# EPICS autosave request: pixciApp/Db/Pixci_settings.req
(P)$(R)TriggerMode
$(P)$(R)SoftTrigger
$(P)$(R)TriggerPolarity
$(P)$(R)UpdateTemperature
$(P)$(R)ToggleTEC
$(P)$(R)ToggleGain
file "ADBase_settings.req", P=$(P), R=$(R)
